PROGRAM POU
VAR
	up_inside: BOOL;
	door_up: BOOL;
	motor_up: BOOL;
	down_inside: BOOL;
	door_down: BOOL;
	motor_down: BOOL;
	motor_off: BOOL;
	key: BOOL;
	up_outside: BOOL;
	down_outside: BOOL;
	TON_0 : TON;
	TON0_et: TIME;
	TON_1: TON;	
	TON1_et: Time;
END_VAR
VAR // added by the converter: edge detectors and wires of the graphical bodies
    _w1, _w2, _w3, _w4, _w5, _w6 : BOOL;
END_VAR

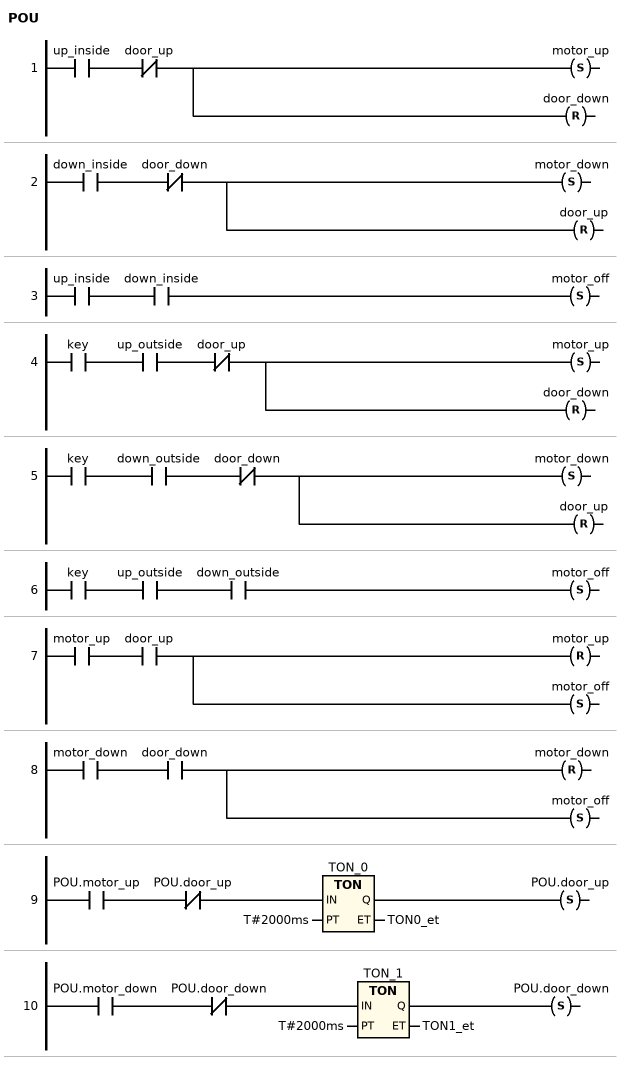
// NETWORK 1
_w1 := up_inside AND NOT door_up;
motor_up S= _w1;
door_down R= _w1;

// NETWORK 2
_w2 := down_inside AND NOT door_down;
motor_down S= _w2;
door_up R= _w2;

// NETWORK 3
motor_off S= up_inside AND down_inside;

// NETWORK 4
_w3 := key AND up_outside AND NOT door_up;
motor_up S= _w3;
door_down R= _w3;

// NETWORK 5
_w4 := key AND down_outside AND NOT door_down;
motor_down S= _w4;
door_up R= _w4;

// NETWORK 6
motor_off S= key AND up_outside AND down_outside;

// NETWORK 7
_w5 := motor_up AND door_up;
motor_up R= _w5;
motor_off S= _w5;

// NETWORK 8
_w6 := motor_down AND door_down;
motor_down R= _w6;
motor_off S= _w6;

// NETWORK 9
TON_0(IN := POU.motor_up AND NOT POU.door_up, PT := T#2000ms, ET => TON0_et); // TON
POU.door_up S= TON_0.Q;

// NETWORK 10
TON_1(IN := POU.motor_down AND NOT POU.door_down, PT := T#2000ms, ET => TON1_et); // TON
POU.door_down S= TON_1.Q;

END_PROGRAM

(* stored: Version 1.1.0.1, ProductVersion 3.1.4022.7
   POU POU: Id {09900206-f166-43e3-a2b8-5c80b0b8b665}, SpecialFunc None *)
